(* PLC project BasePackCtrlX.project, Rexroth ctrlX PLC Engineering ctrlX PLC 1.20.7 *)
(* stored: creationDateTime 2024-08-29T13:23:34.0708601, modificationDateTime 2024-08-29T13:19:13.9101649 *)

(* List of PackTags based on ISA–TR88.00.02-2022 www.hevs.ch Institut Systemes Industriels / Power & Control Project: Automation Box CtrlX S3 Author: Romain Ferrari & Cedric Lenoir Date: 2024 July 31 *)
TYPE HEVS_PackTag_Admin : STRUCT
  Parameter_Real : ARRAY[1..HEVS_PackTag_GVL.C_ADMIN_MAXREALPARAMS] OF HEVS_PackTag_Parameter_Real;
  Parameter_String : ARRAY[1..HEVS_PackTag_GVL.C_ADMIN_MAXSTRINGPARAMS] OF HEVS_PackTag_Parameter_String;
  Parameter_Lreal : ARRAY[1..HEVS_PackTag_GVL.C_ADMIN_MAXLREALPARAMS] OF HEVS_PackTag_Parameter_Lreal;
  Parameter_Dint : ARRAY[1..HEVS_PackTag_GVL.C_ADMIN_MAXDINTPARAMS] OF HEVS_PackTag_Parameter_Dint;
  Alarm : ARRAY[1..HEVS_PackTag_GVL.C_ADMIN_MAXALARMS] OF HEVS_PackTag_Alarm;
  AlarmExtent : DINT;
  AlarmHistory : ARRAY[1..HEVS_PackTag_GVL.C_ADMIN_MAXHISTORYALARMS] OF HEVS_PackTag_Event;
  AlarmHistoryExtent : DINT;
  StopReason : HEVS_PackTag_Event;
  Warning : ARRAY[1..HEVS_PackTag_GVL.C_ADMIN_MAXWARNINGS] OF HEVS_PackTag_Event;
  WarningExtent : DINT;
  ModeTimeCurrent : DINT;
  StateTimeCurrent : DINT;
  CumulativeTime : ARRAY[1..HEVS_PackTag_GVL.C_ADMIN_MAXCUMULATIVETIMES] OF HEVS_PackTag_CumulativeTimes;
  ProductData : ARRAY[1..HEVS_PackTag_GVL.C_ADMIN_MAXPRODUCTDATA] OF HEVS_PackTag_ProductData;
  MachDesignSpeed : REAL;
  DisabledStatesCfg : ARRAY[1..HEVS_PackTag_GVL.C_ADMIN_MAXDISABLEDSTATES] OF DWORD;
  CurDisabledStates : DWORD;
  EnabledModesCfg : DWORD;
  ModeTransitionCfg : ARRAY[1..HEVS_PackTag_GVL.C_ADMIN_MAXMODESTRANSITION] OF DWORD;
  PLCDateTime : HEVS_PackTag_DateTime;
END_STRUCT;
END_TYPE

(* List of PackTags based on ISA–TR88.00.02-2022 www.hevs.ch Institut Systemes Industriels / Power & Control Project: Automation Box CtrlX S3 Author: Romain Ferrari & Cedric Lenoir Date: 2024 July 31 *)
TYPE HEVS_PackTag_Alarm : STRUCT
  Trigger : BOOL;
  ID : DINT;
  Value : DINT;
  Message : STRING;
  Category : DINT;
  DateTime : HEVS_PackTag_DateTime;
  AckDateTime : HEVS_PackTag_DateTime;
END_STRUCT;
END_TYPE

(* List of PackTags based on ISA–TR88.00.02-2022 www.hevs.ch Institut Systemes Industriels / Power & Control Project: Automation Box CtrlX S3 Author: Romain Ferrari & Cedric Lenoir Date: 2024 July 31 *)
TYPE HEVS_PackTag_Command : STRUCT
  UnitMode : DINT;
  UnitModeChangeRequest : BOOL;
  MachSpeed : REAL;
  MaterialIntelock : DWORD;
  CntrlCmd : DINT;
  CmdChangeRequest : BOOL;
  Parameter_Real : ARRAY[1..HEVS_PackTag_GVL.C_COMMAND_MAXSTRINGPARAMS] OF HEVS_PackTag_Parameter_Real;
  Parameter_String : ARRAY[1..HEVS_PackTag_GVL.C_COMMAND_MAXREALPARAMS] OF HEVS_PackTag_Parameter_String;
  Parameter_Lreal : ARRAY[1..HEVS_PackTag_GVL.C_COMMAND_MAXLREALPARAMS] OF HEVS_PackTag_Parameter_Lreal;
  Parameter_Dint : ARRAY[1..HEVS_PackTag_GVL.C_COMMAND_MAXDINTPARAMS] OF HEVS_PackTag_Parameter_Dint;
  SelectedRecipe : DINT;
  RecipeChangeRequest : BOOL;
  Recipe : ARRAY[1..HEVS_PackTag_GVL.C_COMMAND_MAXRECIPE] OF HEVS_PackTag_Recipe;
END_STRUCT;
END_TYPE

(* List of PackTags based on ISA-TR88.00.02-2022 www.hevs.ch Institut Systemes Industriels / Power & Control Project: Automation Box CtrlX S3 Author: Romain Ferrari & Cedric Lenoir Date: 2024 July 30 *)
TYPE HEVS_PackTag_Ingredients : STRUCT
  Parameter_Real : ARRAY[1..HEVS_PackTag_GVL.C_MAXREALINGREDIENTS] OF HEVS_PackTag_Parameter_Real;
  Parameter_String : ARRAY[1..HEVS_PackTag_GVL.C_MAXSTRINGINGREDIENTS] OF HEVS_PackTag_Parameter_String;
  Parameter_Lreal : ARRAY[1..HEVS_PackTag_GVL.C_MAXLREALINGREDIENTS] OF HEVS_PackTag_Parameter_Lreal;
  Parameter_Dint : ARRAY[1...HEVS_PackTag_GVL.C_MAXDINTINGREDIENTS] OF HEVS_PackTag_Parameter_Dint;
END_STRUCT;
END_TYPE

(* List of PackTags based on ISA–TR88.00.02-2022 www.hevs.ch Institut Systemes Industriels / Power & Control Project: Automation Box CtrlX S3 Author: Romain Ferrari & Cedric Lenoir Date: 2024 July 31 *)
TYPE HEVS_PackTag_Status : STRUCT
  UnitModeCurrent : DINT;
  UnitModeRequested : DINT;  (* I consider that there is an error in TR88 2022 §7.5.2.2 *)
  UnitModeChangeInProcess : BOOL;
  StateCurrent : DINT;
  StateRequested : DINT;
  StateChangeInProcess : BOOL;
  MachSpeed : REAL;
  CurMachSpeed : REAL;
  MaterialInterlock : DWORD;
  EquipmentInterlock : HEVS_PackTag_Equipment_Interlock;
  Parameter_Real : ARRAY[1..HEVS_PackTag_GVL.C_STATUS_MAXREALPARAMS] OF HEVS_PackTag_Parameter_Real;
  Parameter_String : ARRAY[1..HEVS_PackTag_GVL.C_STATUS_MAXSTRINGPARAMS] OF HEVS_PackTag_Parameter_String;
  Parameter_Lreal : ARRAY[1..HEVS_PackTag_GVL.C_STATUS_MAXLREALPARAMS] OF HEVS_PackTag_Parameter_Lreal;
  Parameter_Dint : ARRAY[1...HEVS_PackTag_GVL.C_STATUS_MAXDINTPARAMS] OF HEVS_PackTag_Parameter_Dint;
  RecipeCurrent : DINT;
  RecipeRequested : DINT;
  RecipeChangeInProcess : BOOL;
  Recipe : ARRAY[1..HEVS_PackTag_GVL.C_STATUS_MAXRECIPE] OF HEVS_PackTag_Recipe;
  Stacklight : ARRAY[1..HEVS_PackTag_GVL.C_STATUS_MAXSTACKLIGHT] OF DWORD;
END_STRUCT;
END_TYPE

(* List of PackTags based on ISA–TR88.00.02-2022 www.hevs.ch Institut Systemes Industriels / Power & Control Project: Automation Box CtrlX S3 Author: Romain Ferrari & Cedric Lenoir Date: 2024 July 31 *)
TYPE HEVS_PackTag_V2022 : STRUCT
  Command : HEVS_PackTag_Command;
  Status : HEVS_PackTag_Status;
  Admin : HEVS_PackTag_Admin;
END_STRUCT;
END_TYPE

(* www.hevs.ch Institut Systemes Industriels Project: HEVS Pack 2022 Author: Cedric Lenoir Date: 2024 August 29 This structure is made to be available in GVL PackTag With name hevsUI to help diagnositic and interface of this implementation To avoid to lose links if code is modified for info not in base PackTag *)
TYPE HEVS_PackTag_UI : STRUCT
  uiCmdReset : BOOL;  (* Bool commands for UI User inteface *)
  uiCmdStart : BOOL;
  uiCmdStop : BOOL;
  uiCmdHold : BOOL;
  uiCmdUnhold : BOOL;
  uiCmdSuspend : BOOL;
  uiCmdUnsuspend : BOOL;
  uiCmdAbort : BOOL;
  uiCmdClear : BOOL;
  uiCmdComplete : BOOL;
  uiStateClearing : BOOL;  (* Bool states for UI User Inteface *)
  uiStateStopped : BOOL;
  uiStateStarting : BOOL;
  uiStateIdle : BOOL;
  uiStateSuspended : BOOL;
  uiStateExecute : BOOL;
  uiStateStopping : BOOL;
  uiStateAborting : BOOL;
  uiStateAborted : BOOL;
  uiStateHolding : BOOL;
  uiStateHeld : BOOL;
  uiStateUnholding : BOOL;
  uiStateSuspending : BOOL;
  uiStateUnsuspending : BOOL;
  uiStateResetting : BOOL;
  uiStateCompleting : BOOL;
  uiStateCompleted : BOOL;
  uiModeProduction : BOOL;  (* Some Modes of UI User Interface *)
  uiModeMaintenance : BOOL;
  uiModeManual : BOOL;
  uiModeTest : BOOL;
  uiModeUser_05 : BOOL;
  uiModeUser_06 : BOOL;
  uiModeUser_07 : BOOL;
  uiModeUser_08 : BOOL;
  uiStateMasterCurrent : STRING := 'Not linked';  (* Some strings for diagnostic *)
  uiStateMasterDiagnostic : STRING := 'Not linked';
  uiModeMasterCurrent : STRING := 'Not linked';
  uiModeMasterDiagnostic : STRING := 'Not linked';
END_STRUCT;
END_TYPE

(* List of PackTags based on ISA–TR88.00.02-2022 www.hevs.ch Institut Systemes Industriels / Power & Control Project: Automation Box CtrlX S3 Author: Romain Ferrari & Cedric Lenoir Date: 2024 July 30 *)
TYPE HEVS_PackTag_DateTime : STRUCT
  Year : DINT;  (* Can be changed to SINT, INT, or DINT only!! *)
  Month : DINT;  (* Can be changed to SINT, INT, or DINT only!! *)
  Day : DINT;  (* Can be changed to SINT, INT, or DINT only!! *)
  Hour : DINT;  (* Can be changed to SINT, INT, or DINT only!! *)
  Minute : DINT;  (* Can be changed to SINT, INT, or DINT only!! *)
  Second : DINT;  (* Can be changed to SINT, INT, or DINT only!! *)
END_STRUCT;
END_TYPE

(* List of PackTags based on ISA–TR88.00.02-2022 www.hevs.ch Institut Systemes Industriels / Power & Control Project: Automation Box CtrlX S3 Author: Romain Ferrari & Cedric Lenoir Date: 2024 July 30 *)
TYPE HEVS_PackTag_Parameter_Real : STRUCT
  ID : DINT;
  Name : STRING;
  Unit : STRING(6);
  Value : DINT;
END_STRUCT;
END_TYPE

(* List of PackTags based on ISA–TR88.00.02-2022 www.hevs.ch Institut Systemes Industriels / Power & Control Project: Automation Box CtrlX S3 Author: Romain Ferrari & Cedric Lenoir Date: 2024 July 30 *)
TYPE HEVS_PackTag_Parameter_String : STRUCT
  ID : DINT;
  Name : STRING;
  Unit : STRING(6);
  Value : STRING;
END_STRUCT;
END_TYPE

(* List of PackTags based on ISA–TR88.00.02-2022 www.hevs.ch Institut Systemes Industriels / Power & Control Project: Automation Box CtrlX S3 Author: Romain Ferrari & Cedric Lenoir Date: 2024 July 30 *)
TYPE HEVS_PackTag_Parameter_Lreal : STRUCT
  ID : DINT;
  Name : STRING;
  Unit : STRING(6);
  Value : LREAL;
END_STRUCT;
END_TYPE

(* List of PackTags based on ISA–TR88.00.02-2022 www.hevs.ch Institut Systemes Industriels / Power & Control Project: Automation Box CtrlX S3 Author: Romain Ferrari & Cedric Lenoir Date: 2024 July 30 *)
TYPE HEVS_PackTag_Parameter_Dint : STRUCT
  ID : DINT;
  Name : STRING;
  Unit : STRING(6);
  Value : DINT;
END_STRUCT;
END_TYPE

(* List of PackTags based on ISA–TR88.00.02-2022 www.hevs.ch Institut Systemes Industriels / Power & Control Project: Automation Box CtrlX S3 Author: Romain Ferrari & Cedric Lenoir Date: 2024 July 30 *)
TYPE HEVS_PackTag_Recipe : STRUCT
  ID : DINT;
  Name : STRING;
  Unit : STRING(6);
  PrimaryQty : REAL;
  ProcessVariables : HEVS_PackTag_Process_Variables;
  Ingredients : HEVS_PackTag_Ingredients;
END_STRUCT;
END_TYPE

(* List of PackTags based on ISA–TR88.00.02-2022 www.hevs.ch Institut Systemes Industriels / Power & Control Project: Automation Box CtrlX S3 Author: Romain Ferrari & Cedric Lenoir Date: 2024 July 31 *)
TYPE HEVS_PackTag_ProductData : STRUCT
  ID : DINT;
  Name : STRING;
  Unit : STRING(6);
  PrimaryQty : REAL;
  ConsumedCount : DINT;
  ProcessedCount : DINT;
  DefectiveCount : DINT;
  AccConsumedCount : DINT;
  AccProcessedCount : DINT;
  AccDefectiveCount : DINT;
END_STRUCT;
END_TYPE

(* List of PackTags based on ISA–TR88.00.02-2022 www.hevs.ch Institut Systemes Industriels / Power & Control Project: Automation Box CtrlX S3 Author: Romain Ferrari & Cedric Lenoir Date: 2024 July 30 *)
TYPE HEVS_PackTag_CumulativeTimes : STRUCT
  AccTimeSinceReset : DINT;
  ModeStateTimes : ARRAY[0..HEVS_PackTag_GVL.C_MAXMODSTATESTIMES] OF HEVS_PackTag_ModeStateTimes;
END_STRUCT;
END_TYPE

(* List of PackTags based on ISA–TR88.00.02-2022 www.hevs.ch Institut Systemes Industriels / Power & Control Project: Automation Box CtrlX S3 Author: Romain Ferrari & Cedric Lenoir Date: 2024 July 30 *)
TYPE HEVS_PackTag_ModeStateTimes : STRUCT
  Mode : DINT;
  State : ARRAY[0..HEVS_PackTag_GVL.C_MAXSTATES] OF DINT;
END_STRUCT;
END_TYPE

(* List of PackTags based on ISA–TR88.00.02-2022 www.hevs.ch Institut Systemes Industriels / Power & Control Project: Automation Box CtrlX S3 Author: Romain Ferrari & Cedric Lenoir Date: 2024 July 30 *)
TYPE HEVS_PackTag_Process_Variables : STRUCT
  Parameter_Real : ARRAY[1..HEVS_PackTag_GVL.C_MAXREALVARIABLES] OF HEVS_PackTag_Parameter_Real;
  Parameter_String : ARRAY[1..HEVS_PackTag_GVL.C_MAXSTRINGVARIABLES] OF HEVS_PackTag_Parameter_String;
  Parameter_Lreal : ARRAY[1..HEVS_PackTag_GVL.C_MAXLREALVARIABLES] OF HEVS_PackTag_Parameter_Lreal;
  Parameter_Dint : ARRAY[1...HEVS_PackTag_GVL.C_MAXDINTVARIABLES] OF HEVS_PackTag_Parameter_Dint;
END_STRUCT;
END_TYPE

(* List of PackTags based on ISA-TR88.00.02-2022 www.hevs.ch Institut Systemes Industriels / Power & Control Project: Automation Box CtrlX S3 Author: Romain Ferrari & Cedric Lenoir Date: 2024 July 30 *)
TYPE HEVS_PackTag_Event : STRUCT
  Trigger : BOOL;
  ID : DINT;
  Value : DINT;
  Message : STRING;
  Category : DINT;
  DateTime : HEVS_PackTag_DateTime;
  AckDateTime : HEVS_PackTag_DateTime;
END_STRUCT;
END_TYPE

(* List of PackTags based on ISA-TR88.00.02-2022 www.hevs.ch Institut Systemes Industriels / Power & Control Project: Automation Box CtrlX S3 Author: Romain Ferrari & Cedric Lenoir Date: 2024 July 30 *)
TYPE HEVS_PackTag_Equipment_Interlock : STRUCT
  Blocked : BOOL;
  Starved : BOOL;
END_STRUCT;
END_TYPE

(* List of PackTags based on ISA–TR88.00.02-2022 www.hevs.ch Institut Systemes Industriels / Power & Control Project: Automation Box CtrlX S3 Author: Romain Ferrari & Cedric Lenoir Date: 2024 July 31 *)
TYPE HEVS_Min_PackTag_V2022 : STRUCT
  MinCommand : HEVS_Min_PackTag_Command;
  MinStatus : HEVS_Min_PackTag_Status;
  MinAdmin : HEVS_Min_PackTag_Admin;
END_STRUCT;
END_TYPE

(* List of PackTags based on ISA–TR88.00.02-2022 www.hevs.ch Institut Systemes Industriels / Power & Control Project: Automation Box CtrlX S3 Author: Romain Ferrari & Cedric Lenoir Date: 2024 July 31 *)
TYPE HEVS_Min_PackTag_Admin : STRUCT
  ProductData : ARRAY[1..HEVS_PackTag_GVL.C_ADMIN_MAXPRODUCTDATA] OF HEVS_Min_PackTag_ProductData;
  StopReasonMin : HEVS_Min_PackTag_Event;
  CurDisabledStates : DWORD;
END_STRUCT;
END_TYPE

(* List of PackTags based on ISA–TR88.00.02-2022 www.hevs.ch Institut Systemes Industriels / Power & Control Project: Automation Box CtrlX S3 Author: Romain Ferrari & Cedric Lenoir Date: 2024 July 31 *)
TYPE HEVS_Min_PackTag_Command : STRUCT
  UnitMode : DINT;
  UnitModeChangeRequest : BOOL;
  MachSpeed : REAL;
  CntrlCmd : DINT;
  CmdChangeRequest : BOOL;
END_STRUCT;
END_TYPE

(* List of PackTags based on ISA–TR88.00.02-2022 www.hevs.ch Institut Systemes Industriels / Power & Control Project: Automation Box CtrlX S3 Author: Romain Ferrari & Cedric Lenoir Date: 2024 July 31 *)
TYPE HEVS_Min_PackTag_Status : STRUCT
  UnitModeCurrent : DINT;
  StateCurrent : DINT;
  MachSpeed : REAL;
  CurMachSpeed : REAL;
END_STRUCT;
END_TYPE

(* List of PackTags based on ISA–TR88.00.02-2022 www.hevs.ch Institut Systemes Industriels / Power & Control Project: Automation Box CtrlX S3 Author: Romain Ferrari & Cedric Lenoir Date: 2024 July 31 *)
TYPE HEVS_Min_PackTag_ProductData : STRUCT
  ProcessedCount : DINT;
  DefectiveCount : DINT;
END_STRUCT;
END_TYPE

(* List of PackTags based on ISA-TR88.00.02-2022 www.hevs.ch Institut Systemes Industriels / Power & Control Project: Automation Box CtrlX S3 Author: Romain Ferrari & Cedric Lenoir Date: 2024 July 30 *)
TYPE HEVS_Min_PackTag_Event : STRUCT
  ID : DINT;
END_STRUCT;
END_TYPE

(* www.hevs.ch Institut Systemes Industriels Project: Automation Box CtrlX S3 Author: Romain Ferrari Date: 2024 August 16 Summary: Enum OF possible Commands for the Command.CntrlCmd to take. This enum use data type and value according Document: ISA-TR88.00.02-2022 / 7.5.1.5 Command.CntrlCmd Note: Accoring to ISA-TR88.00.02-2022 This is a DINT {attribute 'strict'} *)
{attribute 'qualified_only'}
TYPE E_PackCmd : (eUndefined := 0, eReset := 1, eStart := 2, eStop := 3, eHold := 4, eUnhold := 5, eSuspend := 6, eUnsuspend := 7, eAbort := 8, eClear := 9, eComplete := 10) DINT;
END_TYPE

(* www.hevs.ch Institut Systemes Industriels Project: Automation Box CtrlX S3 Author: Romain Ferrari Date: 2024 August 16 Summary: Enum of possible states for Status.StateCurrent to take. This enum use data type and value according Document: ISA-TR88.00.02-2022 / 7.5.2.4 Status.StateCurrent Note: Accoring to ISA-TR88.00.02-2022 This is a DINT {attribute 'strict'} *)
{attribute 'qualified_only'}
TYPE E_PackState : (eUndefined := 0, eClearing := 1, eStopped := 2, eStarting := 3, eIdle := 4, eSuspended := 5, eExecute := 6, eStopping := 7, eAborting := 8, eAborted := 9, eHolding := 10, eHeld := 11, eUnholding := 12, eSuspending := 13, eUnsuspending := 14, eResetting := 15, eCompleting := 16, eCompleted := 17) DINT;
END_TYPE

(* www.hevs.ch Institut Systemes Industriels Project: HEVS Pack 2022 Author: Cedric Lenoir Date: 2023 October 16 Summary: This enum use data type and value according Document: ISA-TR88.00.02-2022 / 7.5.2.4 State Current Note: Accoring to ISA-TR88.00.02-2022 This is a DINT *)
TYPE ST_PackCmd : STRUCT
  Undefined : BOOL;
  Reset : BOOL;
  Start : BOOL;
  Stop : BOOL;
  Hold : BOOL;
  Unhold : BOOL;
  Suspend : BOOL;
  Unsuspend : BOOL;
  Abort : BOOL;
  Clear : BOOL;
  Complete : BOOL;
  NotUsed : ARRAY[1..14] OF BOOL;
END_STRUCT;
END_TYPE

(* www.hevs.ch Institut Systemes Industriels Project: HEVS Pack 2022 Author: Cedric Lenoir Date: 2024 August 29 This struct is mainly used to build U_StateBitDword *)
TYPE ST_PackState : STRUCT
  Undefined : BIT;
  Clearing : BIT;
  Stopped : BIT;
  Starting : BIT;
  Idle : BIT;
  Suspended : BIT;
  Execute : BIT;
  Stopping : BIT;
  Aborting : BIT;
  Aborted : BIT;
  Holding : BIT;
  Held : BIT;
  Unholding : BIT;
  Suspending : BIT;
  Unsuspending : BIT;
  Resetting : BIT;
  Completing : BIT;
  Completed : BIT;
END_STRUCT;
END_TYPE

(* www.hevs.ch Institut Systemes Industriels Project: Automation Box CtrlX S3 Author: Romain Ferrari Date: 2024 August 16 Summary: Enum of possible modes that Command.UnitMode can take. This enum use data type and value according to Document: ISA-TR88.00.02-2022 / 7.5.1.1 Command.UnitMode Note: Accoring to ISA-TR88.00.02-2022 This is a DINT {attribute 'strict'}: *)
{attribute 'qualified_only'}
TYPE E_PackModes : (Invalid := 0, Production := 1, Maintenance := 2, Manual := 3, Test := 4, User_05 := 5, User_06 := 6, User_07 := 7, User_08 := 8) DINT;
END_TYPE

(* www.hevs.ch Institut Systemes Industriels Project: Automation Box CtrlX S3 Author: Romain Ferrari Date: 2024 August 16 Summary: Enum of possible states that can be disabled using their values in CurDisabledStates. This enum use data type and value according Document: ISA-TR88.00.02-2022 / 7.5.3.22 Admin.CurDisabledStates Note: Accoring to ISA-TR88.00.02-2022 This is a DWORD {attribute 'strict'} *)
{attribute 'qualified_only'}
TYPE E_PackDisabledStates : (none := 0, eClearing := 2, eStopped := 4, eStarting := 8, eIdle := 16, eSuspended := 32, eExecute := 64, eStopping := 128, eAborting := 256, eAborted := 512, eHolding := 1024, eHeld := 2048, eUnholding := 4096, eSuspending := 8192, eUnsuspending := 16384, eResetting := 32768, eCompleting := 65536, eCompleted := 131072) DWORD;
END_TYPE

(* values of E_PackStopReasonId: AbortCondition3: Rename depending the usage; StopCondition3: Rename depending the usage; HoldCondition2: Rename depending the usage; SuspendCondition1: Rename depending the usage; SuspendCondition2: Rename depending the usage More possible states can be added *)

(* www.hevs.ch Institut Systemes Industriels Project: Automation Box CtrlX S3 Author: Romain Ferrari Date: 2024 August 16 Summary: Enum OF possible Commands for the Command_CntrlCmd to take. This enum use data type and value according, but new ID's can be added. Document: ISA-TR88.00.02-2022 / 7.5.3.9.2 StopReason.ID Note: Accoring to ISA-TR88.00.02-2022 This is a DINT {attribute 'strict'} *)
{attribute 'qualified_only'}
TYPE E_PackStopReasonId : (Undefined := 0, RealEstopButtonPushed := 1, VirtualAbortButtonPushed := 2, AbortCondition3 := 3, RealStopButtonPushed := 4, VirtualStopButtonPushed := 5, StopCondition3 := 6, VirtualHoldButtonPushed := 7, HoldCondition2 := 8, SuspendCondition1 := 9, SuspendCondition2 := 10) DINT;
END_TYPE

(* www.hevs.ch Institut Systemes Industriels Project: HEVS Pack 2022 Author: Cedric Lenoir Date: 2024 August 29 This struct is mainly used to build U_ModeBitDword *)
TYPE ST_PackMode : STRUCT
  Invalid : BIT;
  Production : BIT;
  Maintenance : BIT;
  Manual : BIT;
  Test : BIT;
  UserDefinable_5 : BIT;
  UserDefinable_6 : BIT;
  UserDefinable_7 : BIT;
  UserDefinable_8 : BIT;
  UserDefinable_9 : BIT;
  UserDefinable_10 : BIT;
  UserDefinable_11 : BIT;
  UserDefinable_12 : BIT;
  UserDefinable_13 : BIT;
  UserDefinable_14 : BIT;
  UserDefinable_15 : BIT;
  UserDefinable_16 : BIT;
  UserDefinable_17 : BIT;
  UserDefinable_18 : BIT;
  UserDefinable_19 : BIT;
  UserDefinable_20 : BIT;
  UserDefinable_21 : BIT;
  UserDefinable_22 : BIT;
  UserDefinable_23 : BIT;
  UserDefinable_24 : BIT;
  UserDefinable_25 : BIT;
  UserDefinable_26 : BIT;
  UserDefinable_27 : BIT;
  UserDefinable_28 : BIT;
  UserDefinable_29 : BIT;
  UserDefinable_30 : BIT;
  UserDefinable_31 : BIT;
END_STRUCT;
END_TYPE

{attribute 'qualified_only'}
VAR_GLOBAL CONSTANT  (* HEVS_PackTag_GVL - List of PackTags based on ISA–TR88.00.02-2022 www.hevs.ch Institut Systemes Industriels / Power & Control Project: Automation Box CtrlX S3 Author: Romain Ferrari & Cedric Lenoir Date: 2024 July 31 !!!!!! The value of these constants have to be set by the user depending on the system it is implemented on. !!!!!!\\ *)
  C_MAXSTATES : INT := 17;  (* Used in different HEVS_PackML FBs and STRUCTs and in lower branches of the HEVS_PackTag_V30 *)
  C_COMMAND_MAXREALPARAMS : INT := 8;
  C_COMMAND_MAXSTRINGPARAMS : INT := 2;  (* / *)
  C_COMMAND_MAXLREALPARAMS : INT := 8;  (* Used in one of the main PackTag branch of the HEVS_PackTag_V30 : Command *)
  C_COMMAND_MAXDINTPARAMS : INT := 8;
  C_COMMAND_MAXRECIPE : INT := 8;
  C_STATUS_MAXREALPARAMS : INT := 8;  (* / *)
  C_STATUS_MAXSTRINGPARAMS : INT := 2;  (* / *)
  C_STATUS_MAXLREALPARAMS : INT := 8;
  C_STATUS_MAXDINTPARAMS : INT := 8;  (* Used in one of the main PackTag branch of the HEVS_PackTag_V30 : Status *)
  C_STATUS_MAXRECIPE : INT := 8;
  C_STATUS_MAXSTACKLIGHT : INT := 8;
  C_ADMIN_MAXREALPARAMS : INT := 8;  (* / *)
  C_ADMIN_MAXSTRINGPARAMS : INT := 2;  (* / *)
  C_ADMIN_MAXLREALPARAMS : INT := 8;
  C_ADMIN_MAXDINTPARAMS : INT := 8;
  C_ADMIN_MAXALARMS : INT := 8;
  C_ADMIN_MAXHISTORYALARMS : INT := 8;  (* Used in one of the main PackTag branch of the HEVS_PackTag_V30 : Admin *)
  C_ADMIN_MAXWARNINGS : INT := 8;
  C_ADMIN_MAXCUMULATIVETIMES : INT := 11;
  C_ADMIN_MAXPRODUCTDATA : INT := 11;
  C_ADMIN_MAXDISABLEDSTATES : INT := 8;
  C_ADMIN_MAXMODESTRANSITION : INT := 8;  (* is absolutely limited by C_ADMIN_MAXMODESTRANSITIONPACK *)
  C_ADMIN_MAXMODESTRANSITIONPACK : INT := 31;  (* as Pack used DWORD and 0 is reserved, max is limited to 31 *)
  C_MAXMODSTATESTIMES : INT := 8;
  C_MAXREALVARIABLES : INT := 8;
  C_MAXSTRINGVARIABLES : INT := 8;
  C_MAXLREALVARIABLES : INT := 8;
  C_MAXDINTVARIABLES : INT := 8;  (* Used in lower branches of the HEVS_PackTag_V30 *)
  C_MAXREALINGREDIENTS : INT := 8;
  C_MAXSTRINGINGREDIENTS : INT := 8;
  C_MAXLREALINGREDIENTS : INT := 8;
  C_MAXDINTINGREDIENTS : INT := 8;
  hevs_min_packtag_v2022 : HEVS_Min_PackTag_V2022;
END_VAR

{attribute 'qualified_only'}
VAR_GLOBAL  (* PackTag - www.hevs.ch Institut Systemes Industriels Project: HEVS Pack 2022 Author: Cedric Lenoir Date: 2024 August 29 Base GVL for HEVS Pack Tag File name should be PackTag *)
  Command : HEVS_PackTag_Command;
  Status : HEVS_PackTag_Status;
  Admin : HEVS_PackTag_Admin;
  hevsUI : HEVS_PackTag_UI;  (* Help for interface and diagnostic HEVS Pack could be used without this Struc. Can be used with fbCmdBoolInterface Can be used with fbGetActualBoolState *)
END_VAR

TYPE HEVS_Min_PackTag_Union_Dint_FourBytesArray : UNION
  DintAccess : DINT;
  FourBytesArrayAccess : ARRAY[1..4] OF BYTE;
END_UNION;
END_TYPE

TYPE HEVS_Min_PackTag_Union_Dword_Dint_FourBytesArray : UNION
  DwordAccess : DWORD;
  DintAccess : DINT;
  FourBytesArrayAccess : ARRAY[1..4] OF BYTE;
END_UNION;
END_TYPE

TYPE U_StateBitDword : UNION
  dwState : DWORD;
  boolState : ST_PackState;
END_UNION;
END_TYPE

TYPE U_ModeBitDword : UNION
  dwMode : DWORD;
  boolMode : ST_PackMode;
END_UNION;
END_TYPE

(* www.hevs.ch Institut Systemes Industriels Project: HEVS Pack 2022 Author: Cedric Lenoir Date: 2024 August 27 Summary: This FB converts Pack BOOL commnds to Command_CntrlCmd : DINT; Command_CmdChangeRequest : BOOL; Cmd on rising edge only Commands are evaluated with this priority Abort - Stop - Complete - Hold - Suspend - Reset - Clear - Start - Unhold - Unsuspend That means mainly that Abort, then Stop should not be masked by other commands. *)
FUNCTION_BLOCK FB_PackStateCmdBoolInterface
  VAR_INPUT
    Reset : BOOL;
    Start : BOOL;
    Stop : BOOL;
    Hold : BOOL;
    Unhold : BOOL;
    Suspend : BOOL;
    Unsuspend : BOOL;
    Abort : BOOL;
    Clear : BOOL;
    Complete : BOOL;
    remoteEnable : BOOL;  (* For remote, to be completed *)
    remoteCmd : E_PackCmd;
  END_VAR
  VAR_OUTPUT
    eCntrlCmd : E_PackCmd;
    bCmdChangeRequest : BOOL;
  END_VAR
  VAR
    rTrigChangeRequest : R_TRIG;  (* Trigger detect a new command That is, new state is different that last one. *)
    eCntrlCmdMem : E_PackCmd;
    uliTrigCounter : ULINT;  (* For debut, allows to show activation of trigger *)
  END_VAR

            IF Abort THEN
    eCntrlCmd := E_PackCmd.eAbort;
ELSIF Stop THEN
    eCntrlCmd := E_PackCmd.eStop;
ELSIF Complete THEN 
    eCntrlCmd := E_PackCmd.eComplete;
ELSIF Hold THEN
    eCntrlCmd := E_PackCmd.eHold;
ELSIF Suspend THEN 
    eCntrlCmd := E_PackCmd.eSuspend;
ELSIF Reset THEN
    eCntrlCmd := E_PackCmd.eReset;
ELSIF Clear THEN
    eCntrlCmd := E_PackCmd.eClear;
ELSIF Start THEN
    eCntrlCmd := E_PackCmd.eStart;
ELSIF Unhold THEN
    eCntrlCmd := E_PackCmd.eUnhold;
ELSIF Unsuspend THEN
    eCntrlCmd := E_PackCmd.eUnsuspend;
ELSE
    eCntrlCmd := E_PackCmd.eUndefined;
END_IF

rTrigChangeRequest(CLK := eCntrlCmdMem <> eCntrlCmd);
eCntrlCmdMem := eCntrlCmd;
IF rTrigChangeRequest.Q THEN
    uliTrigCounter := uliTrigCounter + 1;
END_IF

bCmdChangeRequest := rTrigChangeRequest.Q;
          
END_FUNCTION_BLOCK

PROGRAM PLC_PACK
  VAR
    uliCount : ULINT;
    fbCmdBoolInterface : FB_PackStateCmdBoolInterface;
    fbModeBoolInterface : FB_PackModeBoolInterface;
    fbModuleTest : FB_ModuleTest;
    whatSC : BOOL;
    testOtherSC : BOOL := TRUE;  (* By setting this flag to FALSE, SC State Complete is disabled *)
    testUMCC : BOOL := TRUE;  (* By setting this flag to FALSE, Unit Mode Change Complete is disabled *)
    fbPackMaster : FB_PackMasterState;
    fbPackMasterMode : FB_PackMasterMode;
    fbGetActualBoolState : FB_GetActualBoolState;
    Admin_CurDisabledStates : DWORD := 0;
    defaultSettingsDone : BOOL;  (* Default settings for Disabled States, set in ACT_SetDefaultSettings *)
    uListOfModesConfig : U_ModeBitDword;  (* Definition of available modes, to be defined in ACT_DefaultSettings. Check below to define Disable State and Transitions for each mode *)
    uDisabledStatesProduction : U_StateBitDword;  (* Invalid := 0, Production := 1, Maintenance := 2, Manual := 3, Test := 4 *)
    uDisabledStatesMaintenance : U_StateBitDword;
    uDisabledStatesManual : U_StateBitDword;
    uDisabledStatesTest : U_StateBitDword;
    uTransitionsProduction : U_StateBitDword;  (* Default settings for State Trsnsitions, set in ACT_SetDefaultSettings Invalid := 0, Production := 1, Maintenance := 2, Manual := 3, Test := 4 *)
    uTransitionsMaintenance : U_StateBitDword;
    uTransitionsManual : U_StateBitDword;
    uTransitionsTest : U_StateBitDword;
  END_VAR

            uliCount := uliCount + 1;

(*
    Init default transitions and disabled states
*)
ACT_SetDefaultSettings();

(*
    BOOL interface for UI Commands
*)
fbCmdBoolInterface(Reset := PackTag.hevsUI.uiCmdReset,
                   Start := PackTag.hevsUI.uiCmdStart,
                   Stop := PackTag.hevsUI.uiCmdStop,
                   Hold := PackTag.hevsUI.uiCmdHold,
                   Unhold := PackTag.hevsUI.uiCmdUnhold,
                   Suspend := PackTag.hevsUI.uiCmdSuspend,
                   Unsuspend := PackTag.hevsUI.uiCmdUnsuspend,
                   Abort := PackTag.hevsUI.uiCmdAbort,
                   Clear := PackTag.hevsUI.uiCmdClear,
                   Complete := PackTag.hevsUI.uiCmdComplete,
                   // Output to Pack Command
                   eCntrlCmd => PackTag.Command.CntrlCmd,
                   bCmdChangeRequest => PackTag.Command.CmdChangeRequest);
				   
(*
	BOOL interface for UI Modes
*)
fbModeBoolInterface(Production := PackTag.hevsUI.uiModeProduction,
                    Maintenance := PackTag.hevsUI.uiModeMaintenance,
					Manual := PackTag.hevsUI.uiModeManual,
					Test := PackTag.hevsUI.uiModeTest,
					// Get actual mode to reset trigger,
					eActualPackMode := PackTag.Status.UnitModeCurrent,
					// Set output commands
    				eCmdUnitMode => PackTag.Command.UnitMode,
					bCmdUnitModeChangeRequest => PackTag.Command.UnitModeChangeRequest);
									   

(*
	List of modules, theoretically EM, eventually CM
*)
fbModuleTest(Status_StateCurrent := PackTag.Status.StateCurrent);
whatSC := fbModuleTest.SC;

(*
	Manage states and mode.
    Receive a AND of SC of each mocule
*)
// For test, select one of default DisabledStates DINT registers
//PackTag.Admin.CurDisabledStates := uDisabledStatesProduction.dwState;
PackTag.Admin.CurDisabledStates := uDisabledStatesTest.dwState;

fbPackMaster(Enable := TRUE,
			 // Inputs
			 SC_StateComplete := whatSC AND testOtherSC,
             Command_CmdChangeRequest := PackTag.Command.CmdChangeRequest,
	         Command_CntrlCmd := PackTag.Command.CntrlCmd,
			 Admin_CurDisabledStates := PackTag.Admin.CurDisabledStates,
			 // Outputs
             Status_StateCurrent => PackTag.Status.StateCurrent,
			 Status_StateChangeInProcess => PackTag.Status.StateChangeInProcess,
			 Status_StateRequested => PackTag.Status.StateRequested,
			 // To help diagnostic and UI
			 strState => PackTag.hevsUI.uiStateMasterCurrent,
			 strDiagnostic	=> PackTag.hevsUI.uiStateMasterDiagnostic);

fbPackMasterMode(Enable := TRUE,
				 StartupMode := E_PackModes.Production,
				 UMCC_UnitModeChangeComplete := testUMCC,
				 // Command selected Mode
				 Cmd_UnitMode := PackTag.Command.UnitMode,
				 Cmd_UnitModeChangeRequest := PackTag.Command.UnitModeChangeRequest,
				 // Current state, from PackTag (Eventually directly from fbPackMaster.Status_StateCurrent
				 Sts_StateCurrent := PackTag.Status.StateCurrent,
			     // To know if a mode is available.
				 Admin_EnabledModesCfg := uListOfModesConfig.dwMode,
				 // To know available possible transitions
				 Admin_ModeTransitionCfg	:= PackTag.Admin.ModeTransitionCfg,
				 // PackTag Status
				 // Invalid := 0, Production := 1, Maintenance := 2, Manual := 3, Test := 4
				 Sts_UnitModeCurrent => PackTag.Status.UnitModeCurrent, 
				 Sts_UnitModeRequested => PackTag.Status.UnitModeRequested,
				 Sts_UnitModeChangeInProcess => PackTag.Status.UnitModeChangeInProcess,
				 // To help diagnostic and UI
				 stringUnitModeCurrent => PackTag.hevsUI.uiModeMasterCurrent,
				 stringModeInfo	=> PackTag.hevsUI.uiModeMasterDiagnostic);	
             
fbGetActualBoolState(Enable := TRUE,
                     ePackState := PackTag.Status.StateCurrent,
                     Clearing => PackTag.hevsUI.uiStateClearing,
                     Stopped => PackTag.hevsUI.uiStateStopped,
                     Starting => PackTag.hevsUI.uiStateStarting,
                     Idle => PackTag.hevsUI.uiStateIdle,
                     Suspended => PackTag.hevsUI.uiStateSuspended,
                     Execute => PackTag.hevsUI.uiStateExecute,
                     Stopping => PackTag.hevsUI.uiStateStopping,
                     Aborting => PackTag.hevsUI.uiStateAborting,
                     Aborted => PackTag.hevsUI.uiStateAborted,
                     Holding => PackTag.hevsUI.uiStateHolding,
                     Held => PackTag.hevsUI.uiStateHeld,
                     Unholding => PackTag.hevsUI.uiStateUnholding,
                     Suspending => PackTag.hevsUI.uiStateSuspending,
                     Unsuspending => PackTag.hevsUI.uiStateUnsuspending,
                     Resetting => PackTag.hevsUI.uiStateResetting,
                     Completing => PackTag.hevsUI.uiStateCompleting,
                     Completed => PackTag.hevsUI.uiStateCompleted);     

          

ACTION ACT_SetDefaultSettings:
                IF NOT defaultSettingsDone THEN
	// Todo only once
	defaultSettingsDone := TRUE;
	(*
		Define list of available modes
		Check C_ADMIN_MAXMODESTRANSITION too.
	*)
	uListOfModesConfig.boolMode.Invalid := FALSE;
	uListOfModesConfig.boolMode.Maintenance := TRUE;
	uListOfModesConfig.boolMode.Manual := TRUE;
	uListOfModesConfig.boolMode.Production := TRUE;
	uListOfModesConfig.boolMode.Test := TRUE;
	uListOfModesConfig.boolMode.UserDefinable_5 := FALSE;
	uListOfModesConfig.boolMode.UserDefinable_6 := FALSE;
	uListOfModesConfig.boolMode.UserDefinable_7 := FALSE;
	uListOfModesConfig.boolMode.UserDefinable_8 := FALSE;

    (*
        A value of 1 in a certain bit location indicates that
        the corresponding state number is disabled.
        
        Init disabled states in Production
    *)
    uDisabledStatesProduction.boolState.Aborted := FALSE;
    uDisabledStatesProduction.boolState.Aborting := FALSE;
    uDisabledStatesProduction.boolState.Clearing := FALSE;
    uDisabledStatesProduction.boolState.Completed := FALSE;
    uDisabledStatesProduction.boolState.Completing := FALSE;
    uDisabledStatesProduction.boolState.Execute := FALSE;
    uDisabledStatesProduction.boolState.Held := FALSE;
    uDisabledStatesProduction.boolState.Holding := FALSE;
    uDisabledStatesProduction.boolState.Unholding := FALSE;
    uDisabledStatesProduction.boolState.Idle := FALSE;
    uDisabledStatesProduction.boolState.Resetting := FALSE;
    uDisabledStatesProduction.boolState.Starting := FALSE;
    uDisabledStatesProduction.boolState.Stopped := FALSE;
    uDisabledStatesProduction.boolState.Stopping := FALSE;
    uDisabledStatesProduction.boolState.Suspended := FALSE;
    uDisabledStatesProduction.boolState.Suspending := FALSE;
    uDisabledStatesProduction.boolState.Unsuspending := FALSE;
    // For Maintenance
    uDisabledStatesMaintenance.boolState.Aborted := FALSE;
    uDisabledStatesMaintenance.boolState.Aborting := FALSE;
    uDisabledStatesMaintenance.boolState.Clearing := TRUE;
    uDisabledStatesMaintenance.boolState.Completed := TRUE;
    uDisabledStatesMaintenance.boolState.Completing := TRUE;
    uDisabledStatesMaintenance.boolState.Execute := FALSE;
    uDisabledStatesMaintenance.boolState.Held := FALSE;
    uDisabledStatesMaintenance.boolState.Holding := FALSE;
    uDisabledStatesMaintenance.boolState.Unholding := FALSE;
    uDisabledStatesMaintenance.boolState.Idle := FALSE;
    uDisabledStatesMaintenance.boolState.Resetting := FALSE;
    uDisabledStatesMaintenance.boolState.Starting := FALSE;
    uDisabledStatesMaintenance.boolState.Stopped := FALSE;
    uDisabledStatesMaintenance.boolState.Stopping := FALSE;
    uDisabledStatesMaintenance.boolState.Suspended := TRUE;
    uDisabledStatesMaintenance.boolState.Suspending := TRUE;
    uDisabledStatesMaintenance.boolState.Unsuspending := TRUE;
    // For Manual
    uDisabledStatesManual.boolState.Aborted := FALSE;
    uDisabledStatesManual.boolState.Aborting := FALSE;
    uDisabledStatesManual.boolState.Clearing := FALSE;
    uDisabledStatesManual.boolState.Completed := TRUE;
    uDisabledStatesManual.boolState.Completing := TRUE;
    uDisabledStatesManual.boolState.Execute := FALSE;
    uDisabledStatesManual.boolState.Held := TRUE;
    uDisabledStatesManual.boolState.Holding := TRUE;
    uDisabledStatesManual.boolState.Unholding := TRUE;
    uDisabledStatesManual.boolState.Idle := FALSE;
    uDisabledStatesManual.boolState.Resetting := FALSE;
    uDisabledStatesManual.boolState.Starting := TRUE;
    uDisabledStatesManual.boolState.Stopped := FALSE;
    uDisabledStatesManual.boolState.Stopping := FALSE;
    uDisabledStatesManual.boolState.Suspended := TRUE;
    uDisabledStatesManual.boolState.Suspending := TRUE;
    uDisabledStatesManual.boolState.Unsuspending := TRUE;
    // For various test
    uDisabledStatesTest.boolState.Aborted := FALSE;
    uDisabledStatesTest.boolState.Aborting := FALSE;
    uDisabledStatesTest.boolState.Clearing := TRUE;
    uDisabledStatesTest.boolState.Completed := FALSE;
    uDisabledStatesTest.boolState.Completing := FALSE;
    uDisabledStatesTest.boolState.Execute := FALSE;
    uDisabledStatesTest.boolState.Held := FALSE;
    uDisabledStatesTest.boolState.Holding := FALSE;
    uDisabledStatesTest.boolState.Unholding := FALSE;
    uDisabledStatesTest.boolState.Idle := FALSE;
    uDisabledStatesTest.boolState.Resetting := FALSE;
    uDisabledStatesTest.boolState.Starting := FALSE;
    uDisabledStatesTest.boolState.Stopped := FALSE;
    uDisabledStatesTest.boolState.Stopping := FALSE;
    uDisabledStatesTest.boolState.Suspended := FALSE;
    uDisabledStatesTest.boolState.Suspending := FALSE;
    uDisabledStatesTest.boolState.Unsuspending := FALSE;
    
    (*
        A value of 1 in a bit location indicates that a mode 
        transition FROM the corresponding state number is allowed
        
        Init transition states in Production
    *)
    uTransitionsProduction.boolState.Aborted := TRUE;
    uTransitionsProduction.boolState.Aborting := FALSE;
    uTransitionsProduction.boolState.Clearing := FALSE;
    uTransitionsProduction.boolState.Completed := TRUE;
    uTransitionsProduction.boolState.Completing := FALSE;
    uTransitionsProduction.boolState.Execute := FALSE;
    uTransitionsProduction.boolState.Held := TRUE;
    uTransitionsProduction.boolState.Holding := FALSE;
    uTransitionsProduction.boolState.Unholding := FALSE;
    uTransitionsProduction.boolState.Idle := FALSE;
    uTransitionsProduction.boolState.Resetting := FALSE;
    uTransitionsProduction.boolState.Starting := FALSE;
    uTransitionsProduction.boolState.Stopped := TRUE;
    uTransitionsProduction.boolState.Stopping := FALSE;
    uTransitionsProduction.boolState.Suspended := FALSE;
    uTransitionsProduction.boolState.Suspending := FALSE;
    uTransitionsProduction.boolState.Unsuspending := FALSE;
    // For Maintenance
    uTransitionsMaintenance.boolState.Aborted := TRUE;
    uTransitionsMaintenance.boolState.Aborting := FALSE;
    uTransitionsMaintenance.boolState.Clearing := FALSE;
    uTransitionsMaintenance.boolState.Completed := FALSE;
    uTransitionsMaintenance.boolState.Completing := FALSE;
    uTransitionsMaintenance.boolState.Execute := FALSE;
    uTransitionsMaintenance.boolState.Held := TRUE;
    uTransitionsMaintenance.boolState.Holding := FALSE;
    uTransitionsMaintenance.boolState.Unholding := FALSE;
    uTransitionsMaintenance.boolState.Idle := FALSE;
    uTransitionsMaintenance.boolState.Resetting := FALSE;
    uTransitionsMaintenance.boolState.Starting := FALSE;
    uTransitionsMaintenance.boolState.Stopped := TRUE;
    uTransitionsMaintenance.boolState.Stopping := FALSE;
    uTransitionsMaintenance.boolState.Suspended := FALSE;
    uTransitionsMaintenance.boolState.Suspending := FALSE;
    uTransitionsMaintenance.boolState.Unsuspending := FALSE;
    // For Manual Mode
    uTransitionsManual.boolState.Aborted := TRUE;
    uTransitionsManual.boolState.Aborting := FALSE;
    uTransitionsManual.boolState.Clearing := FALSE;
    uTransitionsManual.boolState.Completed := FALSE;
    uTransitionsManual.boolState.Completing := FALSE;
    uTransitionsManual.boolState.Execute := FALSE;
    uTransitionsManual.boolState.Held := FALSE;
    uTransitionsManual.boolState.Holding := FALSE;
    uTransitionsManual.boolState.Unholding := FALSE;
    uTransitionsManual.boolState.Idle := TRUE;
    uTransitionsManual.boolState.Resetting := FALSE;
    uTransitionsManual.boolState.Starting := FALSE;
    uTransitionsManual.boolState.Stopped := TRUE;
    uTransitionsManual.boolState.Stopping := FALSE;
    uTransitionsManual.boolState.Suspended := FALSE;
    uTransitionsManual.boolState.Suspending := FALSE;
    uTransitionsManual.boolState.Unsuspending := FALSE;
    // For Test Mode
    uTransitionsTest.boolState.Aborted := TRUE;
    uTransitionsTest.boolState.Aborting := FALSE;
    uTransitionsTest.boolState.Clearing := FALSE;
    uTransitionsTest.boolState.Completed := TRUE;
    uTransitionsTest.boolState.Completing := FALSE;
    uTransitionsTest.boolState.Execute := FALSE;
    uTransitionsTest.boolState.Held := FALSE;
    uTransitionsTest.boolState.Holding := FALSE;
    uTransitionsTest.boolState.Unholding := FALSE;
    uTransitionsTest.boolState.Idle := FALSE;
    uTransitionsTest.boolState.Resetting := FALSE;
    uTransitionsTest.boolState.Starting := FALSE;
    uTransitionsTest.boolState.Stopped := TRUE;
    uTransitionsTest.boolState.Stopping := FALSE;
    uTransitionsTest.boolState.Suspended := FALSE;
    uTransitionsTest.boolState.Suspending := FALSE;
    uTransitionsTest.boolState.Unsuspending := FALSE;

    (*
        Init PackTag
        Invalid := 0, Production := 1, Maintenance := 2, Manual := 3, Test := 4
    *)
    PackTag.Admin.DisabledStatesCfg[1] := uDisabledStatesProduction.dwState;
    PackTag.Admin.DisabledStatesCfg[2] := uDisabledStatesMaintenance.dwState;
    PackTag.Admin.DisabledStatesCfg[3] := uDisabledStatesManual.dwState;
    PackTag.Admin.DisabledStatesCfg[4] := uDisabledStatesTest.dwState;
   
    PackTag.Admin.ModeTransitionCfg[1] := uTransitionsProduction.dwState;
    PackTag.Admin.ModeTransitionCfg[2] := uTransitionsMaintenance.dwState;
    PackTag.Admin.ModeTransitionCfg[3] := uTransitionsManual.dwState;
    PackTag.Admin.ModeTransitionCfg[4] := uTransitionsTest.dwState;
END_IF
              
END_ACTION
END_PROGRAM

(* www.hevs.ch Institut Systemes Industriels Project: HEVS Pack 2022 Author: Cedric Lenoir Date: 2024 August 29 Summary: This FB converts Pack BOOL commnds to Cmd_UnitMode : DINT; Cmd_UnitModeChangeRequest : BOOL; Cmd on rising edge only Modes are evaluated with this priority Production - Maintenance - Manual - Test - User_05 - User_06 - User_07 - User_08 *)
FUNCTION_BLOCK FB_PackModeBoolInterface
  VAR_INPUT
    Production : BOOL;
    Maintenance : BOOL;
    Manual : BOOL;
    Test : BOOL;
    User_05 : BOOL;
    User_06 : BOOL;
    User_07 : BOOL;
    User_08 : BOOL;
    eActualPackMode : E_PackModes;  (* Check change *)
    remoteEnable : BOOL;  (* For remote, to be completed *)
    remoteMode : E_PackModes;
  END_VAR
  VAR_OUTPUT
    eCmdUnitMode : E_PackModes;
    bCmdUnitModeChangeRequest : BOOL;
  END_VAR
  VAR
    waitCycle : UDINT;  (* Trigger detect a new Change Mode That is, new mode is difference than the old one. Delay bCmdUnitModeChangeRequest of one cycle, beause new mode MUST be present before change request *)
    uliTrigCounter : ULINT;  (* For debut, allows to show activation of trigger *)
    timeToResetCommand_ms : INT := 3000;  (* Reset command if no change after 3000 ms *)
    timerToResetCommand : TON;
  END_VAR
  VAR CONSTANT
    C_WAIT_CYCLE : UDINT := 3;
  END_VAR

            IF Production THEN
    eCmdUnitMode := E_PackModes.Production;
ELSIF Maintenance THEN
    eCmdUnitMode := E_PackModes.Maintenance;
ELSIF Manual THEN 
    eCmdUnitMode := E_PackModes.Manual;
ELSIF Test THEN
    eCmdUnitMode := E_PackModes.Test;
ELSIF User_05 THEN 
    eCmdUnitMode := E_PackModes.User_05;
ELSIF User_06 THEN
    eCmdUnitMode := E_PackModes.User_06;
ELSIF User_07 THEN
    eCmdUnitMode := E_PackModes.User_07;
ELSIF User_08 THEN
    eCmdUnitMode := E_PackModes.User_08;
ELSE
	// Invalid, do not set invalid mode at output
    eCmdUnitMode := E_PackModes.Invalid;
END_IF

// Do not process invalid mode
IF NOT (eCmdUnitMode = E_PackModes.Invalid) THEN
	// Do not process if cmd is actual mode.
	IF eActualPackMode = eCmdUnitMode THEN
		bCmdUnitModeChangeRequest := FALSE;
		waitCycle := 0;
	ELSE // Mean eCmdUnitMode is new
		waitCycle := waitCycle + 1;
		IF waitCycle > C_WAIT_CYCLE THEN
			bCmdUnitModeChangeRequest := TRUE;
			// Diagnostic, call of change request
			uliTrigCounter := uliTrigCounter + 1;
		END_IF
	END_IF
END_IF

// Reset command after some time if not possible to change mode.
timerToResetCommand(IN := bCmdUnitModeChangeRequest,
                    PT := INT_TO_TIME(timeToResetCommand_ms));

IF timerToResetCommand.Q THEN
	// Time for change elapsed, command rejected
	// Could be No Valid transition bit
	bCmdUnitModeChangeRequest := FALSE;
END_IF
 

          
END_FUNCTION_BLOCK

(* www.hevs.ch Institut Systemes Industriels Project: HEVS Pack 2022 Author: Cedric Lenoir Date: 2024 August 06 Summary: Used to test and simulate first version of PackMaster Does nothing in Waitstates Wait 2.5 secoond before to return SC in *)
FUNCTION_BLOCK FB_ModuleTest
  VAR_IN_OUT
    Status_StateCurrent : DINT;  (* has to take the PackTag Status.StateCurrent *)
  END_VAR
  VAR
    stateLastCycie : E_PackState := E_PackState.eUndefined;  (* Store last cycle at the en of FB call to detect and state change Used to force minimum of one testSC.In = 0 and reset SC once between each SC *)
    actualState : E_PackState := E_PackState.eAborted;
    init : BOOL;
    testSC : TON;
  END_VAR

            IF NOT init THEN
    init := TRUE;
END_IF

actualState := Status_StateCurrent;

CASE actualState OF
    E_PackState.eUndefined      :;
    E_PackState.eClearing       :;  // Acting
    E_PackState.eStopped        :;
    E_PackState.eStarting       :;  // Acting
    E_PackState.eIdle           :;
    E_PackState.eSuspended      :;
    E_PackState.eExecute        :;  // Acting
    E_PackState.eStopping       :;  // Acting
    E_PackState.eAborting       :;  // Acting
    E_PackState.eAborted        :;
    E_PackState.eHolding        :;  // Acting
    E_PackState.eHeld           :;
    E_PackState.eUnholding      :;  // Acting
    E_PackState.eSuspending     :;  // Acting
    E_PackState.eUnsuspending   :;  // Acting
    E_PackState.eResetting      :;  // Acting
    E_PackState.eCompleting     :;  // Acting
    E_PackState.eCompleted      :;
END_CASE

testSC(IN :=((actualState = E_PackState.eClearing)      OR
             (actualState = E_PackState.eStarting)      OR
             (actualState = E_PackState.eExecute)       OR
             (actualState = E_PackState.eStopping)      OR
             (actualState = E_PackState.eAborting)      OR
             (actualState = E_PackState.eHolding)       OR
             (actualState = E_PackState.eUnholding)     OR
             (actualState = E_PackState.eSuspending)    OR
             (actualState = E_PackState.eUnsuspending)  OR
             (actualState = E_PackState.eResetting)     OR
             (actualState = E_PackState.eCompleting)) AND
             (stateLastCycie = actualState),
        PT := T#2500MS); 
           
stateLastCycie := actualState;
          

PROPERTY SC : BOOL
GET
                    SC := testSC.Q;
                  
END_GET
END_PROPERTY
END_FUNCTION_BLOCK

FUNCTION_BLOCK FB_PackMasterState
  VAR_INPUT
    Enable : BOOL;
    SC_StateComplete : BOOL;  (* Current Acting state of each module is finished. *)
    Command_CntrlCmd : DINT;
    Command_CmdChangeRequest : BOOL;
    Admin_CurDisabledStates : DWORD := 0;  (* In 32 bits, list of disabled states, by default: 0 *)
  END_VAR
  VAR_OUTPUT
    Active : BOOL;
    Status_StateRequested : DINT;
    Status_StateChangeInProcess : BOOL;
    Status_StateCurrent : DINT;
    timeOut : BOOL;  (* TRUE if SC State Complete not present for more than timeTimeOut Could be used for a Warning. *)
    strState : STRING := 'FB not Active';  (* For UI diagnostic and info *)
    strDiagnostic : STRING := 'FB not active';
  END_VAR
  VAR
    masterState : E_PackState := E_PackState.eAborted;
    cntrlCmd : E_PackCmd;
    localDisabledStates : U_StateBitDword;  (* Used to clean Admin_CurDisabledStates if needed. That is, remove acting states if the linked wait state is not present. Use a Union Variant of DWORD *)
    timeTimeOut_ms : INT := 5000;  (* This timer is used to send some info if SC not present for long time. Time in ms, default 5000 means 5 [s] *)
    timeOutCheck : TON;
  END_VAR

            IF Enable THEN
	IF Command_CmdChangeRequest THEN
		cntrlCmd := Command_CntrlCmd;
	ELSE
		cntrlCmd := E_PackCmd.eUndefined;
	END_IF
	
	(*
		Check Admin_CurDisabledStates
		
		Minimum states : Stopped - Idle - Execute - Aborted
	*)
	localDisabledStates.dwState := Admin_CurDisabledStates;
	// Remove extra states for Hold loop
	IF (localDisabledStates.boolState.Held = 1) THEN
		localDisabledStates.boolState.Holding := 1;
		localDisabledStates.boolState.Unholding := 1;
	END_IF
	// Remove extra states for Suspend loop
	IF (localDisabledStates.boolState.Suspended = 1) THEN
		localDisabledStates.boolState.Suspending := 1;
		localDisabledStates.boolState.Unsuspending := 1;
	END_IF
	// Remove extra states for Complete loop
	IF (localDisabledStates.boolState.Completed = 1) THEN
		localDisabledStates.boolState.Completing := 1;
	END_IF
	
	CASE masterState OF														// Based off Production Mode ISA-TR88.00.02-2022
		E_PackState.eUndefined	:
			strState := 'Not Active';
			;
		E_PackState.eAborting 	:
			strState := 'Aborting';
			IF SC_StateComplete THEN
				masterState := E_PackState.eAborted;
			END_IF
			
		E_PackState.eAborted 	:
			strState := 'Aborted';
			IF cntrlCmd = E_PackCmd.eClear THEN								// Clearing is done by the reset. Look at ISA-TR88.00.02-2022
				masterState := M_SkipDisabledState(baseTransition := E_PackState.eClearing,
												   statedisabled := localDisabledStates.boolState.Clearing = 1,
												   nextWaitState := E_PackState.eStopped);
				// masterState := E_PackState.eClearing;
			END_IF
		
		E_PackState.eClearing 	:
			strState := 'Clearing';
			// E-Stop Active Low
			IF cntrlCmd = E_PackCmd.eAbort THEN
				masterState := M_SkipDisabledState(baseTransition := E_PackState.eAborting,
												   statedisabled := localDisabledStates.boolState.Aborting = 1,
												   nextWaitState := E_PackState.eAborted);			
				// masterState := E_PackState.eAborting;
			ELSIF SC_StateComplete THEN
				masterState := E_PackState.eStopped;	
			END_IF
	
		E_PackState.eStopped 	:
			strState := 'Stopped';
			// E-Stop Active Low
			IF cntrlCmd = E_PackCmd.eAbort THEN
				masterState := M_SkipDisabledState(baseTransition := E_PackState.eAborting,
												   statedisabled := localDisabledStates.boolState.Aborting = 1,
												   nextWaitState := E_PackState.eAborted);			
				// masterState := E_PackState.eAborting;
			ELSIF cntrlCmd = E_PackCmd.eReset THEN
				masterState := M_SkipDisabledState(baseTransition := E_PackState.eResetting,
												   statedisabled := localDisabledStates.boolState.Resetting = 1,
												   nextWaitState := E_PackState.eIdle);			
				
				// masterState := E_PackState.eResetting;
			END_IF
	
		E_PackState.eStopping 	:
			strState := 'Stopping';
			// E-Stop Active Low
			IF cntrlCmd = E_PackCmd.eAbort THEN
				masterState := M_SkipDisabledState(baseTransition := E_PackState.eAborting,
												   statedisabled := localDisabledStates.boolState.Aborting = 1,
												   nextWaitState := E_PackState.eAborted);			
				// masterState := E_PackState.eAborting;
			ELSIF SC_StateComplete THEN
				masterState := E_PackState.eStopped;
			END_IF
	
		E_PackState.eResetting 	:
			strState := 'Resetting';
			// E-Stop Active Low
			IF cntrlCmd = E_PackCmd.eAbort THEN
				masterState := M_SkipDisabledState(baseTransition := E_PackState.eAborting,
												   statedisabled := localDisabledStates.boolState.Aborting = 1,
												   nextWaitState := E_PackState.eAborted);			
				
				// masterState := E_PackState.eAborting;
			ELSIF cntrlCmd = E_PackCmd.eStop THEN
				masterState := M_SkipDisabledState(baseTransition := E_PackState.eStopping,
												   statedisabled := localDisabledStates.boolState.Stopping = 1,
												   nextWaitState := E_PackState.eStopped);	
				// masterState := E_PackState.eStopping;
			ELSIF SC_StateComplete THEN
				masterState := E_PackState.eIdle;			
			END_IF
	
		E_PackState.eIdle 		:
			strState := 'Idle';
			// E-Stop Active Low
			IF cntrlCmd = E_PackCmd.eAbort THEN
				masterState := M_SkipDisabledState(baseTransition := E_PackState.eAborting,
												   statedisabled := localDisabledStates.boolState.Aborting = 1,
												   nextWaitState := E_PackState.eAborted);			
				
				// masterState := E_PackState.eAborting;
			ELSIF cntrlCmd = E_PackCmd.eStop THEN
				masterState := M_SkipDisabledState(baseTransition := E_PackState.eStopping,
												   statedisabled := localDisabledStates.boolState.Stopping = 1,
												   nextWaitState := E_PackState.eStopped);	
				// masterState := E_PackState.eStopping;
			ELSIF cntrlCmd = E_PackCmd.eStart THEN
				masterState := M_SkipDisabledState(baseTransition := E_PackState.eStarting,
												   statedisabled := localDisabledStates.boolState.Starting = 1,
												   nextWaitState := E_PackState.eExecute);	
				
				// masterState := E_PackState.eStarting;
			END_IF
	
		E_PackState.eStarting 	:
			strState := 'Starting';
			// E-Stop Active Low
			IF cntrlCmd = E_PackCmd.eAbort THEN
				masterState := M_SkipDisabledState(baseTransition := E_PackState.eAborting,
												   statedisabled := localDisabledStates.boolState.Aborting = 1,
												   nextWaitState := E_PackState.eAborted);			
				
				// masterState := E_PackState.eAborting;
			ELSIF cntrlCmd = E_PackCmd.eStop THEN
				masterState := M_SkipDisabledState(baseTransition := E_PackState.eStopping,
												   statedisabled := localDisabledStates.boolState.Stopping = 1,
												   nextWaitState := E_PackState.eStopped);	
				
				// masterState := E_PackState.eStopping;
			ELSIF SC_StateComplete THEN
				masterState := E_PackState.eExecute;	
			END_IF
	
		E_PackState.eExecute 	:
			strState := 'Execute';
			// E-Stop Active Low
			IF cntrlCmd = E_PackCmd.eAbort THEN
				masterState := M_SkipDisabledState(baseTransition := E_PackState.eAborting,
												   statedisabled := localDisabledStates.boolState.Aborting = 1,
												   nextWaitState := E_PackState.eAborted);			
				
				// masterState := E_PackState.eAborting;
			ELSIF cntrlCmd = E_PackCmd.eStop THEN
				masterState := M_SkipDisabledState(baseTransition := E_PackState.eStopping,
												   statedisabled := localDisabledStates.boolState.Stopping = 1,
												   nextWaitState := E_PackState.eStopped);	
				
				// masterState := E_PackState.eStopping;
			ELSIF cntrlCmd = E_PackCmd.eHold AND 
				  // If Hold disabled
				  NOT (localDisabledStates.boolState.Held = 1) THEN
				masterState := M_SkipDisabledState(baseTransition := E_PackState.eHolding,
												   statedisabled := localDisabledStates.boolState.Holding = 1,
												   nextWaitState := E_PackState.eHeld);				  
				// masterState := E_PackState.eHolding;	
			ELSIF cntrlCmd = E_PackCmd.eSuspend  AND 
				  // If Suspend disabled
				  NOT (localDisabledStates.boolState.Suspended = 1) THEN
				masterState := M_SkipDisabledState(baseTransition := E_PackState.eSuspending,
												   statedisabled := localDisabledStates.boolState.Suspending = 1,
												   nextWaitState := E_PackState.eSuspended);				  
				// masterState := E_PackState.eSuspending;	
			ELSIF cntrlCmd = E_PackCmd.eComplete AND 
				  // If Completed disabled
				  NOT (localDisabledStates.boolState.Completed = 1) THEN
				masterState := M_SkipDisabledState(baseTransition := E_PackState.eCompleting,
												   statedisabled := localDisabledStates.boolState.Completing = 1,
												   nextWaitState := E_PackState.eCompleted);				  
				// masterState := E_PackState.eCompleting;	
			END_IF
			
			
		(* Held Loop *)
		E_PackState.eHolding	:
			strState := 'Holding';
			// E-Stop Active Low
			IF cntrlCmd = E_PackCmd.eAbort THEN
				masterState := M_SkipDisabledState(baseTransition := E_PackState.eAborting,
												   statedisabled := localDisabledStates.boolState.Aborting = 1,
												   nextWaitState := E_PackState.eAborted);			
				
				// masterState := E_PackState.eAborting;
			ELSIF cntrlCmd = E_PackCmd.eStop THEN
				masterState := M_SkipDisabledState(baseTransition := E_PackState.eStopping,
												   statedisabled := localDisabledStates.boolState.Stopping = 1,
												   nextWaitState := E_PackState.eStopped);	
				
				// masterState := E_PackState.eStopping;
			ELSIF SC_StateComplete THEN
				masterState := E_PackState.eHeld;	
			END_IF
			
		E_PackState.eHeld		:
			strState := 'Held';
			// E-Stop Active Low
			IF cntrlCmd = E_PackCmd.eAbort THEN
				masterState := M_SkipDisabledState(baseTransition := E_PackState.eAborting,
												   statedisabled := localDisabledStates.boolState.Aborting = 1,
												   nextWaitState := E_PackState.eAborted);			
				
				// masterState := E_PackState.eAborting;
			ELSIF cntrlCmd = E_PackCmd.eStop THEN
				masterState := M_SkipDisabledState(baseTransition := E_PackState.eStopping,
												   statedisabled := localDisabledStates.boolState.Stopping = 1,
												   nextWaitState := E_PackState.eStopped);	
				
				// masterState := E_PackState.eCompleting;
			ELSIF cntrlCmd = E_PackCmd.eComplete AND 
				  // If Completed disabled
				  NOT (localDisabledStates.boolState.Completed = 1) THEN
				masterState := M_SkipDisabledState(baseTransition := E_PackState.eCompleting,
												   statedisabled := localDisabledStates.boolState.Completing = 1,
												   nextWaitState := E_PackState.eCompleted);				  
				// masterState := E_PackState.eCompleting;            
			ELSIF cntrlCmd = E_PackCmd.eUnhold THEN
				masterState := M_SkipDisabledState(baseTransition := E_PackState.eUnholding,
												   statedisabled := localDisabledStates.boolState.Unholding = 1,
												   nextWaitState := E_PackState.eExecute);				  
				// masterState := E_PackState.eUnholding;
			END_IF
	
		E_PackState.eUnholding	:
			strState := 'Unholding';
			// E-Stop Active Low
			IF cntrlCmd = E_PackCmd.eAbort THEN
				masterState := M_SkipDisabledState(baseTransition := E_PackState.eAborting,
												   statedisabled := localDisabledStates.boolState.Aborting = 1,
												   nextWaitState := E_PackState.eAborted);			
				
				// masterState := E_PackState.eAborting;
			ELSIF cntrlCmd = E_PackCmd.eStop THEN
				masterState := M_SkipDisabledState(baseTransition := E_PackState.eStopping,
												   statedisabled := localDisabledStates.boolState.Stopping = 1,
												   nextWaitState := E_PackState.eStopped);	
				
				// masterState := E_PackState.eStopping;
			ELSIF SC_StateComplete THEN
				masterState := E_PackState.eExecute;	
			END_IF
			
		E_PackState.eSuspending	:
			strState := 'Suspending';
			// E-Stop Active Low
			IF cntrlCmd = E_PackCmd.eAbort THEN
				masterState := M_SkipDisabledState(baseTransition := E_PackState.eAborting,
												   statedisabled := localDisabledStates.boolState.Aborting = 1,
												   nextWaitState := E_PackState.eAborted);			
				
				// masterState := E_PackState.eAborting;
			ELSIF cntrlCmd = E_PackCmd.eStop THEN
				masterState := M_SkipDisabledState(baseTransition := E_PackState.eStopping,
												   statedisabled := localDisabledStates.boolState.Stopping = 1,
												   nextWaitState := E_PackState.eStopped);	
				
				// masterState := E_PackState.eStopping;
			ELSIF SC_StateComplete THEN
				masterState := E_PackState.eSuspended;	
			END_IF
			
		E_PackState.eUnsuspending	:
			strState := 'Unsuspending';
			// E-Stop Active Low
			IF cntrlCmd = E_PackCmd.eAbort THEN
				masterState := M_SkipDisabledState(baseTransition := E_PackState.eAborting,
												   statedisabled := localDisabledStates.boolState.Aborting = 1,
												   nextWaitState := E_PackState.eAborted);			
				
				// masterState := E_PackState.eAborting;
			ELSIF cntrlCmd = E_PackCmd.eStop THEN
				masterState := M_SkipDisabledState(baseTransition := E_PackState.eStopping,
												   statedisabled := localDisabledStates.boolState.Stopping = 1,
												   nextWaitState := E_PackState.eStopped);	
				
				// masterState := E_PackState.eStopping;
			ELSIF SC_StateComplete THEN
				masterState := E_PackState.eExecute;	
			END_IF
			
		E_PackState.eSuspended	:
			strState := 'Suspended';
			// E-Stop Active Low
			IF cntrlCmd = E_PackCmd.eAbort THEN
				masterState := M_SkipDisabledState(baseTransition := E_PackState.eAborting,
												   statedisabled := localDisabledStates.boolState.Aborting = 1,
												   nextWaitState := E_PackState.eAborted);			
				// masterState := E_PackState.eAborting;
			ELSIF cntrlCmd = E_PackCmd.eStop THEN
				masterState := M_SkipDisabledState(baseTransition := E_PackState.eStopping,
												   statedisabled := localDisabledStates.boolState.Stopping = 1,
												   nextWaitState := E_PackState.eStopped);	
				// masterState := E_PackState.eStopping;
			ELSIF cntrlCmd = E_PackCmd.eComplete AND 
				  // If Completed disabled
				  NOT (localDisabledStates.boolState.Completed = 1) THEN
				masterState := M_SkipDisabledState(baseTransition := E_PackState.eCompleting,
												   statedisabled := localDisabledStates.boolState.Completing = 1,
												   nextWaitState := E_PackState.eCompleted);			
				// masterState := E_PackState.eCompleting;	
			ELSIF cntrlCmd = E_PackCmd.eHold AND 
				  // If Hold disabled
				  NOT (localDisabledStates.boolState.Held = 1) THEN
				masterState := M_SkipDisabledState(baseTransition := E_PackState.eHolding,
												   statedisabled := localDisabledStates.boolState.Holding = 1,
												   nextWaitState := E_PackState.eHeld);			
				// masterState := E_PackState.eHolding;	
			ELSIF cntrlCmd = E_PackCmd.eUnsuspend THEN
				masterState := M_SkipDisabledState(baseTransition := E_PackState.eUnsuspending,
												   statedisabled := localDisabledStates.boolState.Unsuspending = 1,
												   nextWaitState := E_PackState.eExecute);			
				// masterState := E_PackState.eUnsuspending;
			END_IF
			
		E_PackState.eCompleting	:
			strState := 'Completing';
			// E-Stop Active Low
			IF cntrlCmd = E_PackCmd.eAbort THEN
				masterState := M_SkipDisabledState(baseTransition := E_PackState.eAborting,
												   statedisabled := localDisabledStates.boolState.Aborting = 1,
												   nextWaitState := E_PackState.eAborted);			
				
				// masterState := E_PackState.eAborting;
			ELSIF cntrlCmd = E_PackCmd.eStop THEN
				masterState := M_SkipDisabledState(baseTransition := E_PackState.eStopping,
												   statedisabled := localDisabledStates.boolState.Stopping = 1,
												   nextWaitState := E_PackState.eStopped);	
				
				// masterState := E_PackState.eStopping;
			ELSIF SC_StateComplete THEN
				masterState := E_PackState.eCompleted;
			END_IF
			
		E_PackState.eCompleted	:
			strState := 'Completed';
			// E-Stop Active Low
			IF cntrlCmd = E_PackCmd.eAbort THEN
				masterState := M_SkipDisabledState(baseTransition := E_PackState.eAborting,
												   statedisabled := localDisabledStates.boolState.Aborting = 1,
												   nextWaitState := E_PackState.eAborted);			
				
				// masterState := E_PackState.eAborting;
			ELSIF cntrlCmd = E_PackCmd.eStop THEN
				masterState := M_SkipDisabledState(baseTransition := E_PackState.eStopping,
												   statedisabled := localDisabledStates.boolState.Stopping = 1,
												   nextWaitState := E_PackState.eStopped);	
				// masterState := E_PackState.eStopping;
			ELSIF cntrlCmd = E_PackCmd.eReset THEN
				masterState := M_SkipDisabledState(baseTransition := E_PackState.eResetting,
												   statedisabled := localDisabledStates.boolState.Resetting = 1,
												   nextWaitState := E_PackState.eIdle);	
				// masterState := E_PackState.eResetting;
			END_IF
			
	END_CASE
	
	(*
		Set output of FB
	*)
	IF Command_CmdChangeRequest THEN
		Status_StateRequested := Command_CntrlCmd;
	ELSE
		Status_StateRequested := E_PackState.eUndefined;	
	END_IF
	Status_StateChangeInProcess := Command_CmdChangeRequest AND (Status_StateRequested <> Status_StateCurrent);
	Status_StateCurrent := masterState;

	// Check Time out
	timeOutCheck(IN := (masterState = E_PackState.eAborting)   OR
                       (masterState = E_PackState.eClearing)   OR
                       (masterState = E_PackState.eCompleting) OR
                       (masterState = E_PackState.eHolding)    OR
                       (masterState = E_PackState.eResetting)  OR
                       (masterState = E_PackState.eStarting)   OR
                       (masterState = E_PackState.eStopping)   OR
                       (masterState = E_PackState.eSuspending) OR
                       (masterState = E_PackState.eUnholding)  OR
                       (masterState = E_PackState.eUnsuspending),
		         PT := INT_TO_TIME(timeTimeOut_ms));
				 
	IF timeOutCheck.Q THEN
		strDiagnostic := CONCAT('Timeout with: ',strState);
	ELSE
		strDiagnostic := 'No Message';
	END_IF

	Active := TRUE;
ELSE // FB not Enable
	Active := FALSE;
	strState := 'FB not Active';
	strDiagnostic := 'FB not active';	
END_IF

          

METHOD M_SkipDisabledState : E_PackState
  VAR_INPUT
    baseTransition : E_PackState;  (* Next state if statedisabled is FALSE *)
    statedisabled : BOOL;  (* Disabled condition, e.g. (localDisabledStates.boolState.Stopping = 1) *)
    nextWaitState : E_PackState;  (* Next state if statedisabled is TRUE *)
  END_VAR
                  IF NOT statedisabled THEN
	M_SkipDisabledState := baseTransition;
ELSE
	M_SkipDisabledState := nextWaitState;
END_IF
                
END_METHOD
END_FUNCTION_BLOCK

(* www.hevs.ch Institut Systemes Industriels Project: HEVS Pack 2022 Author: Cedric Lenoir Date: 2024 August 27 Summary: This FB return the BOOL State format of: PackTag.Status.StateCurrent *)
FUNCTION_BLOCK FB_GetActualBoolState
  VAR_INPUT
    Enable : BOOL;
    ePackState : E_PackState;
  END_VAR
  VAR_OUTPUT
    Active : BOOL;
    Clearing : BOOL;
    Stopped : BOOL;
    Starting : BOOL;
    Idle : BOOL;
    Suspended : BOOL;
    Execute : BOOL;
    Stopping : BOOL;
    Aborting : BOOL;
    Aborted : BOOL;
    Holding : BOOL;
    Held : BOOL;
    Unholding : BOOL;
    Suspending : BOOL;
    Unsuspending : BOOL;
    Resetting : BOOL;
    Completing : BOOL;
    Completed : BOOL;
  END_VAR

            IF Enable THEN
	Clearing := ePackState = E_PackState.eClearing;
	Stopped := ePackState = E_PackState.eStopped;
	Starting := ePackState = E_PackState.eStarting;
	Idle := ePackState = E_PackState.eIdle;
	Suspended := ePackState = E_PackState.eSuspended;
	Execute := ePackState = E_PackState.eExecute;
	Stopping := ePackState = E_PackState.eStopping;
	Aborting := ePackState = E_PackState.eAborting;
	Aborted := ePackState = E_PackState.eAborted;
	Holding := ePackState = E_PackState.eHolding;
	Held := ePackState = E_PackState.eHeld;
	Unholding := ePackState = E_PackState.eUnholding;
	Suspending := ePackState = E_PackState.eSuspending;
	Unsuspending := ePackState = E_PackState.eUnsuspending;
	Resetting := ePackState = E_PackState.eResetting;
	Completing := ePackState = E_PackState.eCompleting;
	Completed := ePackState = E_PackState.eCompleted;    
ELSE
	Clearing := FALSE;
	Stopped := FALSE;
	Starting := FALSE;
	Idle := FALSE;
	Suspended := FALSE;
	Execute := FALSE;
	Stopping := FALSE;
	Aborting := FALSE;
	Aborted := FALSE;
	Holding := FALSE;
	Held := FALSE;
	Unholding := FALSE;
	Suspending := FALSE;
	Unsuspending := FALSE;
	Resetting := FALSE;
	Completing := FALSE;
	Completed := FALSE;     
END_IF

Active := Enable;
          
END_FUNCTION_BLOCK

(* www.hevs.ch Institut Systemes Industriels Project: HEVS Pack 2022 Author: Cedric Lenoir Date: 2024 August 28 Summary: Mode manager Default at start is Production mode := 1 *)
FUNCTION_BLOCK FB_PackMasterMode
  VAR_INPUT
    Enable : BOOL;
    UMCC_UnitModeChangeComplete : BOOL := TRUE;  (* Unit Mode Change Complete, must be TRUE when all Module have finiched Change. If no delay requested, could be set to TRUE by default *)
    StartupMode : DINT := E_PackModes.Production;  (* Read once at first cycle, cannot be changed later. *)
    Cmd_UnitMode : DINT;  (* Command selected Mode, must be present when Cmd_UnitModeChangeRequest is activated. *)
    Cmd_UnitModeChangeRequest : BOOL;  (* Command is set upon rising edge of the boolean. *)
    Sts_StateCurrent : DINT := E_PackState.eAborted;  (* The actual state is needed to determine if transition is possible in Admin_ModeTransitionCfg *)
    Admin_EnabledModesCfg : DWORD;  (* To know if a mode is available. *)
    Admin_ModeTransitionCfg : ARRAY[1..HEVS_PackTag_GVL.C_ADMIN_MAXMODESTRANSITION] OF DWORD;  (* To know available possible transitions *)
  END_VAR
  VAR_OUTPUT
    Active : BOOL;  (* FB Active *)
    Sts_UnitModeCurrent : DINT;  (* Invalid := 0, Production := 1, Maintenance := 2, Manual := 3, Test := 4 *)
    Sts_UnitModeRequested : DINT;  (* Invalid if not Cmd_UnitModeChangeRequest *)
    Sts_UnitModeChangeInProcess : BOOL;
    stringUnitModeCurrent : STRING;  (* UnitModeCurrent in STRING format Actually set in the code of This FB. *)
    stringModeInfo : STRING;  (* Change mode Help, some info *)
  END_VAR
  VAR
    uliLoop : ULINT;
    currentMode : DINT := E_PackModes.Production;
    bInitDone : BOOL;
    rTrigChangeRequest : R_TRIG;
    internalChangeInProgress : BOOL;  (* Use to maintain change mode until end of change. *)
    stringModeCurrent : ARRAY[0..HEVS_PackTag_GVL.C_ADMIN_MAXMODESTRANSITION] OF STRING := ['Invalid', 'Production', 'Maintenance', 'Manual', 'Test HEVS', 'User 05', 'User 06', 'User 07', 'User 08'];
    uliTriggerChangeRequested : ULINT;  (* For diagnostic *)
    bValidModeFound : BOOL;
    setTestDWord : DWORD;  (* Compute a DWord with exactly one bit *)
    internalCurrentModeEnblTra : BOOL;  (* Current mode enable transition from state *)
    internalTargetModeEnblTra : BOOL;  (* Target mode enable transition to state *)
  END_VAR

            IF Enable THEN
	IF NOT bInitDone THEN
		bInitDone := TRUE;
		currentMode := StartupMode;
		stringUnitModeCurrent := stringModeCurrent[currentMode];
	END_IF
	uliLoop := uliLoop + 1;

	rTrigChangeRequest(clk := Cmd_UnitModeChangeRequest);

	// Main condition to start a change request is Cmd_UnitModeChangeRequest
	// Once the change has started, it is maintained until the change is complete.
	IF rTrigChangeRequest.Q 									  AND 
	   // Change only possible if Cmd_UnitMode < max unit modes, else ignord
	   Cmd_UnitMode < HEVS_PackTag_GVL.C_ADMIN_MAXMODESTRANSITION AND
	   // Cmd_UnitMode MUST NOT be 0
	   Cmd_UnitMode > 0											  AND
	   // Do not process anything if mode is equal to currentMode 
	   Cmd_UnitMode <> currentMode                                AND
	   // Admin.EnabledModesCfg = 1 or less means no valid mode enabled
	   Admin_EnabledModesCfg > 1								  THEN
	   
	   bValidModeFound := TRUE;
	   uliTriggerChangeRequested := uliTriggerChangeRequested + 1;
	   // A valid mode number is available and enabled
	   // Compute test DWORD
	   setTestDWord := 1;
	   setTestDWord := SHL(setTestDWord,Sts_StateCurrent);
	   // For Current mode
	   internalCurrentModeEnblTra := (Admin_ModeTransitionCfg[currentMode] AND setTestDWord) = setTestDWord;
	   // For target mode
	   internalTargetModeEnblTra := (Admin_ModeTransitionCfg[Cmd_UnitMode] AND setTestDWord) = setTestDWord;

	   // Check if there are valid states transitions in Admin_ModeTransitionCfg
	   IF internalCurrentModeEnblTra AND
		  internalTargetModeEnblTra  THEN
			 internalChangeInProgress := TRUE;
			 stringUnitModeCurrent := 'Mode is Changing';
			 stringModeInfo := 'Wait UMCC_UnitModeChangeComplete';
	   ELSE
		   // Do nothing
	      stringModeInfo := 'No valid transition bits';
	   END_IF
		
	   // Check
	ELSIF NOT bValidModeFound THEN
		// Do nothing
		stringModeInfo := 'No valid mode';
    ELSE
		// Do nothing
		;
	END_IF	
	
	// Once internalChangeInProgress is set,
	// wait UMCC_UnitModeChangeComplete for end of mode change.
	IF internalChangeInProgress    AND
	   UMCC_UnitModeChangeComplete THEN
		internalChangeInProgress := FALSE;
		// Update current mode
		currentMode := Cmd_UnitMode;
		stringUnitModeCurrent := stringModeCurrent[currentMode];
		stringModeInfo := 'Mode changed successfully';
	END_IF
	(*
		Manage outputs
	*)
	Active := Enable;
	Sts_UnitModeCurrent := currentMode;
	IF Cmd_UnitModeChangeRequest THEN
		Sts_UnitModeRequested := Cmd_UnitMode;
	ELSE
		Sts_UnitModeRequested := E_PackModes.Invalid;
	END_IF
	Sts_UnitModeChangeInProcess := internalChangeInProgress AND (Cmd_UnitMode <> currentMode);
	
	IF NOT Cmd_UnitModeChangeRequest THEN
		bValidModeFound := FALSE;
		stringModeInfo := 'Wait Cmd_UnitModeChangeRequest';
	END_IF	
ELSE // FB not Enable, reset outputs
	Active := FALSE;
	Sts_UnitModeCurrent := 0;
	Sts_UnitModeRequested := 0;
	Sts_UnitModeChangeInProcess	:= FALSE;
	stringUnitModeCurrent := 'FB Not active';
	// Change mode Help, some info				
	stringModeInfo := 'FB Not active';	
END_IF


          
END_FUNCTION_BLOCK
